(* CODESYS project xlh_dc_motor_simple_00_01.project
   Description: Receives some incoming messages and echoes them with CAN-ID +1
   Company: 3S - Smart Software Solutions GmbH
   Version: 1.0.0.0
   Title: CAN Bus API Example
   Author: 3S - Smart Software Solutions GmbH

Project tree, tasks and I/O mapping:
  xLH_base : CODESYS Control for Raspberry Pi 64 SL, CODESYS, order no. 2302000009, version 4.20.0.0
    application app
      libraries: Standard, 3.5.22.0 (System); Util, 3.5.22.0 (System); VisuDialogs, * (System); Memory, * (3S - Smart Software Solutions GmbH); CmpBitmapPool, * (System); CAN API, 1.0.0.4 (CODESYS); MemoryUtils, * (3S - Smart Software Solutions GmbH); xLH Control Systems, 0.1 (xemax ag); CAA CiA 405, 4.3.0.0 (CODESYS)
      task MAIN_TASK (cyclic, interval 10 ms, priority 1) calls io, MAIN_CALLER
      task VISU_TASK (cyclic, interval 100 ms, priority 31) calls VisuElems.Visu_Prg
      trace Trace_Switch (task MAIN_TASK): MAIN.diEncoderPosition, MAIN.fSpeed, MAIN.fCurrentMa
      program MAIN [CFC]
      visualisation VISU_RET_DCM
      text list TextListForCombobox_eControllerType
      IO/
        program io [ST]
        function block FB_XLH_GPIO [ST]: read, write
      program MAIN_CALLER [ST]
    SoftMotion General Axis Pool
      a_axis : SM_Drive_PosControl, CODESYS, order no. 1805, version 4.18.0.0
          settings: wDriveID = 4; dwRatioTechUnitsDenom = 101846; iRatioTechUnitsNum = -125; eRampType = 1; fSWMaxVelocity = 50; fSWMaxAcceleration = 100; fSWMaxDeceleration = 100; fSWMaxJerk = 1000; fSWLimitNegative = -1000.0; ScalingIncs = 814768; ScalingUnits = 1000; InvertDirection = TRUE; IsLinearMotor = TRUE; MaximumOutputVelocityInt = 40738; MinimumOutputVelocityInt = -40738; Kp = 0.05; MaxFollowingError = 5.0; EnableFollowingErrorCheck = TRUE; DeadTime = 3.0
      x_axis : SM_Drive_PosControl, CODESYS, order no. 1805, version 4.18.0.0
          settings: dwRatioTechUnitsDenom = 101846; iRatioTechUnitsNum = 125; eRampType = 1; fSWMaxVelocity = 50; fSWMaxAcceleration = 100; fSWMaxDeceleration = 100; fSWMaxJerk = 1000; fSWLimitNegative = -1000; ScalingIncs = 814768; ScalingUnits = 1000; IsLinearMotor = TRUE; MaximumOutputVelocityInt = 40738; MinimumOutputVelocityInt = -40738; Kp = 0.05; MaxFollowingError = 5.0; EnableFollowingErrorCheck = TRUE; DeadTime = 3.0
      y_axis : SM_Drive_PosControl, CODESYS, order no. 1805, version 4.18.0.0
          settings: wDriveID = 2; dwRatioTechUnitsDenom = 101846; iRatioTechUnitsNum = 125; eRampType = 1; fSWMaxVelocity = 50; fSWMaxAcceleration = 100; fSWMaxDeceleration = 100; fSWMaxJerk = 1000; fSWLimitNegative = -1000; ScalingIncs = 814768; ScalingUnits = 1000; IsLinearMotor = TRUE; MaximumOutputVelocityInt = 40738; MinimumOutputVelocityInt = -40738; Kp = 0.05; MaxFollowingError = 5.0; EnableFollowingErrorCheck = TRUE; DeadTime = 3.0
      z_axis : SM_Drive_PosControl, CODESYS, order no. 1805, version 4.18.0.0
          settings: wDriveID = 3; dwRatioTechUnitsDenom = 101846; iRatioTechUnitsNum = 125; eRampType = 1; fSWMaxVelocity = 50; fSWMaxAcceleration = 100; fSWMaxDeceleration = 100; fSWMaxJerk = 1000; fSWLimitNegative = -1000; ScalingIncs = 814768; ScalingUnits = 1000; IsLinearMotor = TRUE; MaximumOutputVelocityInt = 40738; MinimumOutputVelocityInt = -40738; Kp = 0.05; MaxFollowingError = 5.0; EnableFollowingErrorCheck = TRUE; DeadTime = 3.0
    GPIOs_A_B : GPIOs B+/Pi2, CODESYS, version 4.20.0.0
        input  app.io.gpio.bSw1 : BOOL  // digital inputs (GPIO0..GPIO31).Bit4
        input  app.io.gpio.bSw2 : BOOL  // digital inputs (GPIO0..GPIO31).Bit5
        input  app.io.gpio.bSw3 : BOOL  // digital inputs (GPIO0..GPIO31).Bit6
        input  app.io.gpio.bSw4 : BOOL  // digital inputs (GPIO0..GPIO31).Bit12
        input  app.io.gpio.bSw5 : BOOL  // digital inputs (GPIO0..GPIO31).Bit13
        input  app.io.gpio.bSw6 : BOOL  // digital inputs (GPIO0..GPIO31).Bit16
        input  app.io.gpio.bSw7 : BOOL  // digital inputs (GPIO0..GPIO31).Bit17
        input  app.io.gpio.bSw8 : BOOL  // digital inputs (GPIO0..GPIO31).Bit19
        output app.io.gpio.bLed1 : BOOL  // digital outputs (GPIO0..GPIO31).Bit20
        output app.io.gpio.bLed2 : BOOL  // digital outputs (GPIO0..GPIO31).Bit21
        output app.io.gpio.bLed3 : BOOL  // digital outputs (GPIO0..GPIO31).Bit22
        output app.io.gpio.bLed4 : BOOL  // digital outputs (GPIO0..GPIO31).Bit23
        output app.io.gpio.bLed5 : BOOL  // digital outputs (GPIO0..GPIO31).Bit24
        output app.io.gpio.bLed6 : BOOL  // digital outputs (GPIO0..GPIO31).Bit26
        output app.io.gpio.bLed7 : BOOL  // digital outputs (GPIO0..GPIO31).Bit27
        unmapped channels: digital inputs (GPIO0..GPIO31), digital outputs (GPIO0..GPIO31)
    Onewire
    Camera device
      <Leer>
    SPI
    I²C
    CANbus : CANbus, CODESYS, version 4.3.0.0
        settings: Baudrate = 1000 kbit/s
      CANopen_Manager : CANopen_Manager, CODESYS, version 4.3.0.0
          settings: ConfigVersion = 50659584
        xlh_dc_motor : xlh_dc_motor, xemax ag, order no. 0, version Revision=16#00000001, FileVersion=1.0
            settings: NODEIDSAVED = 1; SDO Timeout = 1000000; PDO_Autoconfig = FALSE; EXPERTSETTINGS = FALSE; Sync-General Parameters.Sync-COBID = 16#00000080; Sync-General Parameters.Communication Cycle Period = 16#00000000 usec; PDO 16#1400.COBID = 16#00000201; Process by CANopenManager = TRUE; PDO 16#1800.COBID = 16#00000181; Process by CANopenManager = TRUE; Control.Subindex = 16#01; PWM Duty Cycle.Subindex = 16#02; Position.Subindex = 16#01; dt per Increment.Subindex = 16#02; Current.Subindex = 16#01; SDO List.Set COB-ID sync.Index = 16#1005; SDO List.Set COB-ID sync.Subindex = 16#00; SDO List.Set COB-ID sync.Value = 16#00000080; SDO List.Set COB-ID sync.Size = 32; SDO List.Set COB-ID sync.AbortIfError = FALSE; SDO List.Set COB-ID sync.JumpToLine = FALSE; SDO List.Set COB-ID sync.Line = 0; SDO List.Set communication cycle period.Index = 16#1006; SDO List.Set communication cycle period.Subindex = 16#00; SDO List.Set communication cycle period.Value = 16#00000000; SDO List.Set communication cycle period.Size = 32; SDO List.Set communication cycle period.AbortIfError = FALSE; SDO List.Set communication cycle period.JumpToLine = FALSE; SDO List.Set communication cycle period.Line = 0; SDO List.Set Guardtime.Index = 16#100C; SDO List.Set Guardtime.Subindex = 16#00; SDO List.Set Guardtime.Value = 16#000000C8; SDO List.Set Guardtime.Size = 16; SDO List.Set Guardtime.AbortIfError = FALSE; SDO List.Set Guardtime.JumpToLine = FALSE; SDO List.Set Guardtime.Line = 0; SDO List.Set Lifetime.Index = 16#100D; SDO List.Set Lifetime.Subindex = 16#00; SDO List.Set Lifetime.Value = 16#00000003; SDO List.Set Lifetime.Size = 8;
              SDO List.Set Lifetime.AbortIfError = FALSE; SDO List.Set Lifetime.JumpToLine = FALSE; SDO List.Set Lifetime.Line = 0; SDO List.Set Heartbeat Consumer.Index = 16#1016; SDO List.Set Heartbeat Consumer.Subindex = 16#01; SDO List.Set Heartbeat Consumer.Value = 0; SDO List.Set Heartbeat Consumer.Size = 32; SDO List.Set Heartbeat Consumer.AbortIfError = FALSE; SDO List.Set Heartbeat Consumer.JumpToLine = FALSE; SDO List.Set Heartbeat Consumer.Line = 0; SDO List.Disable PDO.Index = 16#1400; SDO List.Disable PDO.Subindex = 16#01; SDO List.Disable PDO.Value = 16#80000201; SDO List.Disable PDO.Size = 32; SDO List.Disable PDO.AbortIfError = FALSE; SDO List.Disable PDO.JumpToLine = FALSE; SDO List.Disable PDO.Line = 0; SDO List.Set transmission type.Index = 16#1400; SDO List.Set transmission type.Subindex = 16#02; SDO List.Set transmission type.Value = 16#FF; SDO List.Set transmission type.Size = 8; SDO List.Set transmission type.AbortIfError = FALSE; SDO List.Set transmission type.JumpToLine = FALSE; SDO List.Set transmission type.Line = 0; SDO List.Set and enable COB-ID.Index = 16#1400; SDO List.Set and enable COB-ID.Subindex = 16#01; SDO List.Set and enable COB-ID.Value = 16#00000201; SDO List.Set and enable COB-ID.Size = 32; SDO List.Set and enable COB-ID.AbortIfError = FALSE; SDO List.Set and enable COB-ID.JumpToLine = FALSE; SDO List.Set and enable COB-ID.Line = 0; SDO List.Disable PDO.Index = 16#1800; SDO List.Disable PDO.Subindex = 16#01; SDO List.Disable PDO.Value = 16#80000181; SDO List.Disable PDO.Size = 32; SDO List.Disable PDO.AbortIfError = FALSE; SDO List.Disable PDO.JumpToLine = FALSE; SDO List.Disable PDO.Line = 0; SDO List.Set transmission type.Index = 16#1800; SDO List.Set transmission type.Subindex = 16#02;
              SDO List.Set transmission type.Value = 16#FF; SDO List.Set transmission type.Size = 8; SDO List.Set transmission type.AbortIfError = FALSE; SDO List.Set transmission type.JumpToLine = FALSE; SDO List.Set transmission type.Line = 0; SDO List.Set inhibit time.Index = 16#1800; SDO List.Set inhibit time.Subindex = 16#03; SDO List.Set inhibit time.Value = 16#0000; SDO List.Set inhibit time.Size = 16; SDO List.Set inhibit time.AbortIfError = FALSE; SDO List.Set inhibit time.JumpToLine = FALSE; SDO List.Set inhibit time.Line = 0; SDO List.Set event time.Index = 16#1800; SDO List.Set event time.Subindex = 16#05; SDO List.Set event time.Value = 16#0000; SDO List.Set event time.Size = 16; SDO List.Set event time.AbortIfError = FALSE; SDO List.Set event time.JumpToLine = FALSE; SDO List.Set event time.Line = 0; SDO List.Set and enable COB-ID.Index = 16#1800; SDO List.Set and enable COB-ID.Subindex = 16#01; SDO List.Set and enable COB-ID.Value = 16#00000181; SDO List.Set and enable COB-ID.Size = 32; SDO List.Set and enable COB-ID.AbortIfError = FALSE; SDO List.Set and enable COB-ID.JumpToLine = FALSE; SDO List.Set and enable COB-ID.Line = 0; ConfigVersion = 50659584
            output app.io.bMotorCcw : BOOL  // Control.Bit0
            output app.io.bMotorCw : BOOL  // Control.Bit1
            output app.io.uiMotorSpeed : UINT  // PWM Duty Cycle
            input  app.io.diEncoderPosition : DINT  // Position
            input  app.io.iEncoderDtInc : INT  // dt per Increment
            input  app.io.uiCurrent : UINT  // Current
            unmapped channels: Control
  libraries: VisuSymbols, 4.5.0.0 (System); DepictorBase, 1.2.0.0 (CODESYS)
  text list GlobalTextList
  5ce3da45-db07-42e7-a21c-a00fff4ed8f6|C:\Users\phe\Downloads\Musterloesung_FUP.PNG
*)

// xLH_base/app/IO/io
PROGRAM io
VAR_INPUT
	gpio: FB_XLH_GPIO;	
	diEncoderPosition: DINT;// CanOpen variable
	iEncoderDtInc: INT;// CanOpen variable
	uiCurrent: UINT;// CanOpen variable
	fMotorDutyCycle: LREAL;// +- 100.0
END_VAR
VAR_OUTPUT
	bMotorCw: BOOL;// CanOpen variable
	bMotorCcw: BOOL;// CanOpen variable
	uiMotorSpeed: UINT;// CanOpen variable
	fSpeed: LREAL;
	fCurrentMa: LREAL;
	bDummy: BOOL;
END_VAR
VAR
	fSpeedTemp: LREAL;
	fbPt2Speed: PT2:= (fK:=1.0, fT1:= 0.020, fT2:= 0.020);
	fbPt2Current: PT2:= (fK:=1.0, fT1:= 0.50, fT2:= 0.50);
END_VAR

// DC Motor 6V => 106 RPM = 1.78 Hz
// DC Motor 5V =>  89 RPM = 1.49 Hz

IF iEncoderDtInc <> 0 THEN
	fSpeedTemp := 1350 / TO_LREAL(iEncoderDtInc) ;
ELSE
	fSpeedTemp := 0.0;
END_IF
fbPt2Speed(fX:=fSpeedTemp, fY=>fSpeed);

fbPt2Current(fX:=TO_LREAL(uiCurrent)/10.0, fY=>fCurrentMa);

IF fMotorDutyCycle >= 0.0 THEN
	bMotorCw := TRUE;
	bMotorCcw := FALSE;
ELSE
	bMotorCw := FALSE;
	bMotorCcw := TRUE;
END_IF
uiMotorSpeed := LREAL_TO_UINT(LIMIT(0.0, ABS(fMotorDutyCycle * 450.0), 45000));

END_PROGRAM

// xLH_base/app/IO/FB_XLH_GPIO
FUNCTION_BLOCK FB_XLH_GPIO
VAR_INPUT
	bLed1: BOOL;
	bLed2: BOOL;
	bLed3: BOOL;
	bLed4: BOOL;
	bLed5: BOOL;
	bLed6: BOOL;
	bLed7: BOOL;	
END_VAR
VAR_OUTPUT
	bSw1: BOOL;
	bSw2: BOOL;
	bSw3: BOOL;
	bSw4: BOOL;
	bSw5: BOOL;
	bSw6: BOOL;
	bSw7: BOOL;
	bSw8: BOOL;
END_VAR

METHOD read : BOOL
VAR_INPUT
END_VAR
END_METHOD

METHOD write : BOOL
VAR_INPUT
END_VAR
END_METHOD

END_FUNCTION_BLOCK

// xLH_base/app/MAIN_CALLER
PROGRAM MAIN_CALLER
VAR
	bDevicesCoRunning: BOOL;
	fbTonDevicesCoRunning: TON := (PT:=T#250MS);
END_VAR

fbTonDevicesCoRunning(IN:= 
	(xlh_dc_motor.CANopenState = _3SCOS.DEVICE_STATE.OPERATIONAL)
);
// if all devices are in RUN status (including delay), POU MAIN is called.
IF fbTonDevicesCoRunning.Q THEN
	MAIN();
END_IF

END_PROGRAM

// xLH_base/app/MAIN
PROGRAM MAIN
VAR
	bControllerEnable: BOOL;
	fSetPoint: LREAL := 1.0;
	fSetPointOffset: LREAL := 0.0;
	fManualDutyCycle: LREAL;
	fbControllerSpeed: Controller := (eTyp := eControllerType.PIDT1, 
                                      fKr := 4.0, 
                                      fTn := 0.05, 
                                      fTv := 0.250, 
                                      fTvz := 0.05);
	fbBlink: Blink := (ENABLE:=TRUE, TIMEHIGH:=T#5S, TIMELOW:=T#5S);
	fW: LREAL;
END_VAR
VAR // added by the converter: edge detectors and wires of the graphical bodies
    _w1 : LREAL;
END_VAR

// task cycle time plc
// The project uses the XlhControlSystems library.
//
// https://github.com/xemax-ag/xLH-applications/tree/main/xlh-control-systems
//
// If this is not installed, it can be added manually under Tools, Library Repository
CS_COMMOM(fDt := 0.010);
// Simple implementation of speed control system
// An optimized version with linearization and data logger modeling in a simulation environment is demonstrated in the
// xlh_dc_motor_advanced_xx_xx.project.
fbBlink(); // Blink
_w1 := SEL(fbBlink.OUT, 0.0, fSetPointOffset) + fSetPoint;
fbControllerSpeed(fE := _w1 - io.fSpeed, bReset := NOT bControllerEnable); // Controller
fW := _w1;
io.fMotorDutyCycle := SEL(bControllerEnable, fManualDutyCycle, fbControllerSpeed.fY);

END_PROGRAM

// xLH_base/app/VISU_RET_DCM
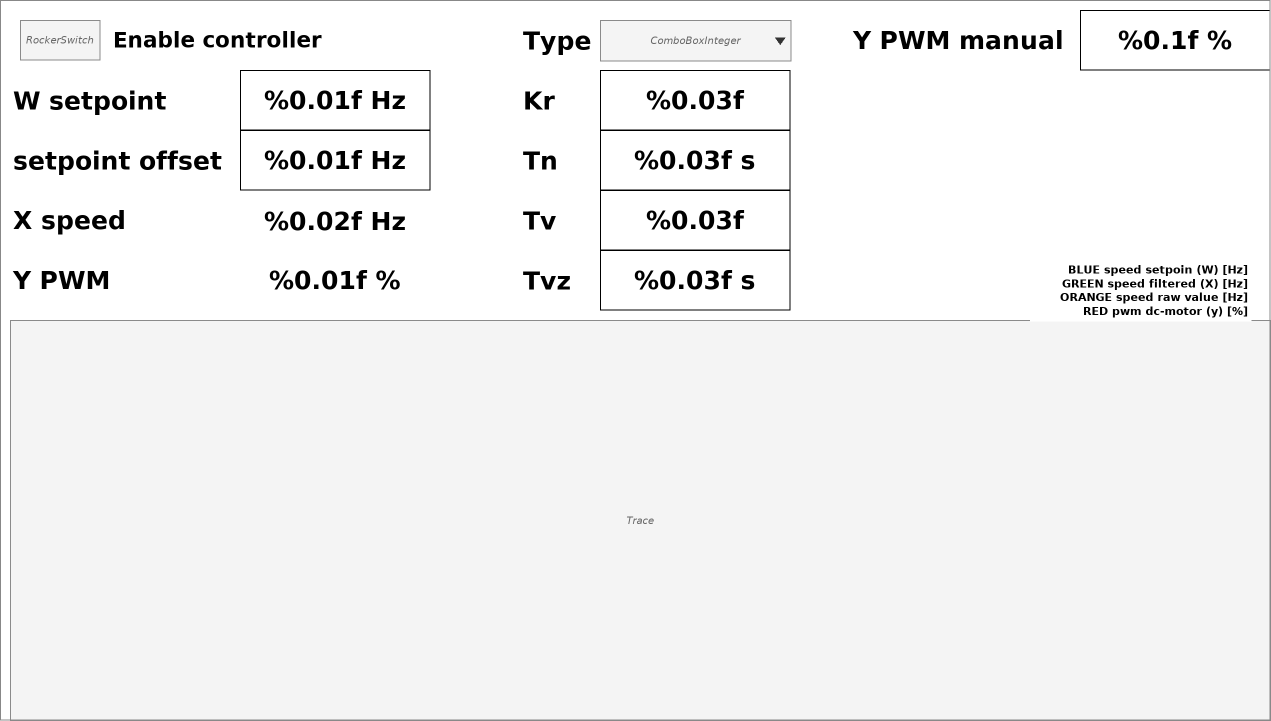
VISUALIZATION VISU_RET_DCM  // 1271x721
    Trace (10,320 1261x401)
    Rectangle (1030,260 221x61), "BLUE speed setpoin (W) [Hz] GREEN speed filtered (X) [Hz] ORANGE speed raw value [Hz] RED pwm dc-motor (y) [%]"
    Rectangle (240,250 190x60), "%0.01f %", text variable: io.fMotorDutyCycle, invisible if: NOT MAIN.bControllerEnable
    Rectangle (10,250 181x60), "Y PWM", invisible if: NOT MAIN.bControllerEnable
        OnMouseClick:  OpenModal=True, PositionX=200, PositionY=100
    Rectangle (10,70 181x61), "W setpoint", invisible if: NOT MAIN.bControllerEnable
        OnMouseClick:  Dialog=Dialog_Signalgenerator_W_Drehzahl, OpenModal=True, PositionX=100, PositionY=100
    Rectangle (240,70 190x60), "%0.01f Hz", text variable: MAIN.fSetPoint, invisible if: NOT MAIN.bControllerEnable
        OnMouseClick: write the text variable via Default
    Rectangle (240,191 190x60), "%0.02f Hz", text variable: io.fSpeed
    Rectangle (10,190 181x60), "X speed"
    Rectangle (110,20 281x40), "Enable controller"
        OnMouseClick:  Dialog=Dialog_Linearisierung_Drehzahl, OpenModal=True, PositionX=100, PositionY=100
    RockerSwitch (20,20 80x40), variable: MAIN.bControllerEnable, behaviour: TOGGLE, style: Switch-RockerSwitch-Gray
    Rectangle (850,10 221x60), "Y PWM manual", invisible if: MAIN.bControllerEnable
        OnMouseClick:  Dialog=Dialog_Signalgenerator_Y, OpenModal=True, PositionX=200, PositionY=100
    Rectangle (1080,10 190x60), "%0.1f %", text variable: MAIN.fManualDutyCycle, invisible if: MAIN.bControllerEnable
        OnMouseClick: write the text variable via Default, min -100.0, max 100.0
    Rectangle (600,70 190x60), "%0.03f", text variable: MAIN.fbControllerSpeed.fKr, invisible if: NOT MAIN.bControllerEnable OR (MAIN.fbControllerSpeed.eTyp = eControllerType.I)
        OnMouseClick: write the text variable via Default
    Rectangle (520,70 80x61), "Kr", invisible if: NOT MAIN.bControllerEnable OR (MAIN.fbControllerSpeed.eTyp = eControllerType.I)
        OnMouseClick:  Dialog=Dialog_Signalgenerator_W_Drehzahl, OpenModal=True, PositionX=100, PositionY=100
    Rectangle (600,130 190x60), "%0.03f s", text variable: MAIN.fbControllerSpeed.fTn, invisible if: NOT MAIN.bControllerEnable OR (MAIN.fbControllerSpeed.eTyp = eControllerType.P) OR (MAIN.fbControllerSpeed.eTyp = eControllerType.PDT1)
        OnMouseClick: write the text variable via Default
    Rectangle (520,130 80x61), "Tn", invisible if: NOT MAIN.bControllerEnable OR (MAIN.fbControllerSpeed.eTyp = eControllerType.P) OR (MAIN.fbControllerSpeed.eTyp = eControllerType.PDT1)
        OnMouseClick:  Dialog=Dialog_Signalgenerator_W_Drehzahl, OpenModal=True, PositionX=100, PositionY=100
    Rectangle (600,190 190x60), "%0.03f", text variable: MAIN.fbControllerSpeed.fTv, invisible if: NOT MAIN.bControllerEnable OR (MAIN.fbControllerSpeed.eTyp = eControllerType.P) OR (MAIN.fbControllerSpeed.eTyp = eControllerType.I) OR (MAIN.fbControllerSpeed.eTyp = eControllerType.PI)
        OnMouseClick: write the text variable via Default
    Rectangle (520,190 80x61), "Tv", invisible if: NOT MAIN.bControllerEnable OR (MAIN.fbControllerSpeed.eTyp = eControllerType.P) OR (MAIN.fbControllerSpeed.eTyp = eControllerType.I) OR (MAIN.fbControllerSpeed.eTyp = eControllerType.PI)
        OnMouseClick:  Dialog=Dialog_Signalgenerator_W_Drehzahl, OpenModal=True, PositionX=100, PositionY=100
    Rectangle (600,250 190x60), "%0.03f s", text variable: MAIN.fbControllerSpeed.fTvz, invisible if: NOT MAIN.bControllerEnable OR (MAIN.fbControllerSpeed.eTyp = eControllerType.P) OR (MAIN.fbControllerSpeed.eTyp = eControllerType.I) OR (MAIN.fbControllerSpeed.eTyp = eControllerType.PI)
        OnMouseClick: write the text variable via Default
    Rectangle (520,250 81x61), "Tvz", invisible if: NOT MAIN.bControllerEnable OR (MAIN.fbControllerSpeed.eTyp = eControllerType.P) OR (MAIN.fbControllerSpeed.eTyp = eControllerType.I) OR (MAIN.fbControllerSpeed.eTyp = eControllerType.PI)
        OnMouseClick:  Dialog=Dialog_Signalgenerator_W_Drehzahl, OpenModal=True, PositionX=100, PositionY=100
    ComboBoxInteger (600,20 191x41), variable: MAIN.fbControllerSpeed.eTyp, invisible if: NOT MAIN.bControllerEnable, text list: 'TextListForCombobox_eControllerType'
    Rectangle (520,10 80x61), "Type", invisible if: NOT MAIN.bControllerEnable
        OnMouseClick:  Dialog=Dialog_Signalgenerator_W_Drehzahl, OpenModal=True, PositionX=100, PositionY=100
    Rectangle (10,130 221x61), "setpoint offset", invisible if: NOT MAIN.bControllerEnable
        OnMouseClick:  Dialog=Dialog_Signalgenerator_W_Drehzahl, OpenModal=True, PositionX=100, PositionY=100
    Rectangle (240,130 190x60), "%0.01f Hz", text variable: MAIN.fSetPointOffset, invisible if: NOT MAIN.bControllerEnable
        OnMouseClick: write the text variable via Default
END_VISUALIZATION

(* text list TextListForCombobox_eControllerType (id | default)
  1 | P
  2 | I
  3 | PI
  4 | PDT1
  5 | PIDT1
   |  *)
